Omron CX-Programmer project NewProject (CX-Programmer 9.75)

# PLC ChemicalMixingTimer: CP1E N30

## Global symbols (name address type ; comment)
T000 BOOL  ; T0
T001 BOOL  ; T1
T002 BOOL  ; T2
T003 BOOL  ; T3

## Program NewProgram1 (cyclic task 0)
Local symbols
MainSupply 100.00 BOOL  ; 100.00
MixingMotor 100.03 BOOL  ; 100.03
Start 0.00 BOOL  ; 0.00
Stop 0.01 BOOL  ; 0.01
V1 100.01 BOOL  ; 100.01
V2 100.02 BOOL  ; 100.02
V3 100.04 BOOL  ; 100.04

### Section Section1

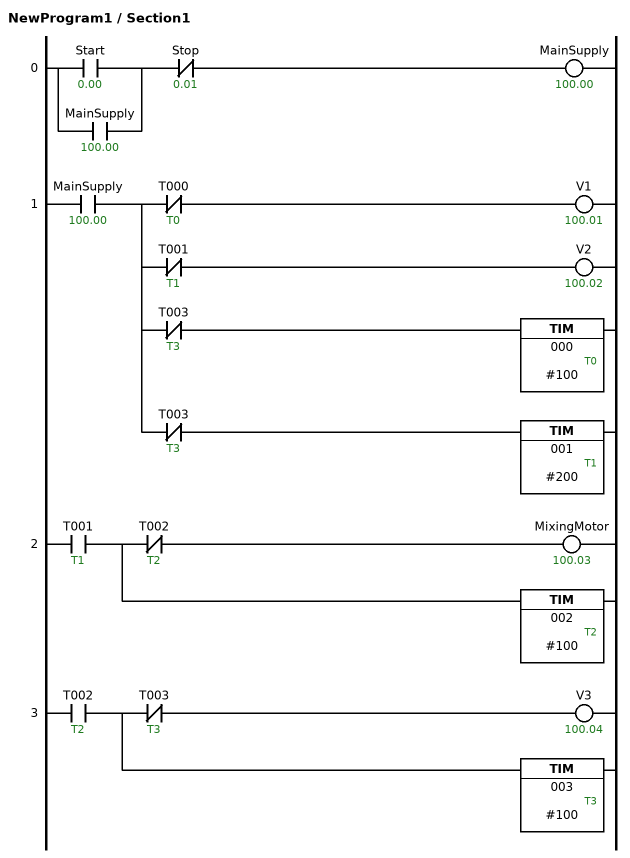
; rung 0
LD Start  ; 0.00
OR MainSupply  ; 100.00
ANDNOT Stop  ; 0.01
OUT MainSupply  ; 100.00
; rung 1
LD MainSupply  ; 100.00
OUT TR0
ANDNOT T000  ; T0
OUT V1  ; 100.01
LD TR0
ANDNOT T001  ; T1
OUT V2  ; 100.02
LD TR0
ANDNOT T003  ; T3
TIM 000 #100  ; T0
LD TR0
ANDNOT T003  ; T3
TIM 001 #200  ; T1
; rung 2
LD T001  ; T1
OUT TR0
ANDNOT T002  ; T2
OUT MixingMotor  ; 100.03
LD TR0
TIM 002 #100  ; T2
; rung 3
LD T002  ; T2
OUT TR0
ANDNOT T003  ; T3
OUT V3  ; 100.04
LD TR0
TIM 003 #100  ; T3

### Section END
; rung 0
END(001)